// TIA Portal V17 program export: 1 tag tables, 0 data types, 0 data blocks, 1 code blocks (in call order from the OBs), 0 instance data blocks

VAR_GLOBAL   // PLC tag table "Default tag table"
   START AT %M0.0 : Bool;
   STOP AT %M0.1 : Bool;
   MOTOR AT %Q0.0 : Bool;
END_VAR

ORGANIZATION_BLOCK "Main"   // OB1, LAD, ProgramCycle
TITLE = "Main Program Sweep (Cycle)"
{ S7_Optimized_Access := 'TRUE' }
VERSION : 0.1
// stored: AutoNumber true, IsIECCheckEnabled false, SetENOAutomatically false
   VAR_INPUT
      Initial_Call : Bool;   // Initial call of this OB
      Remanence : Bool;   // =True, if remanent data are available
   END_VAR
BEGIN

REGION Network 1
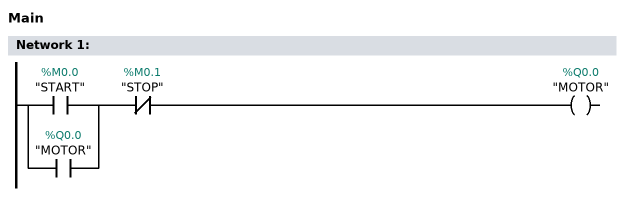
   RUNG wire#powerrail
      Contact( "START" )
      wire#w1
      I_Contact( "STOP" )
      Coil( "MOTOR" )
   END_RUNG
   RUNG wire#powerrail
      Contact( "MOTOR" )
   END_RUNG wire#w1
   // the same network as SCL:
   "MOTOR" := ("START" OR "MOTOR") AND NOT "STOP";
END_REGION
END_ORGANIZATION_BLOCK
